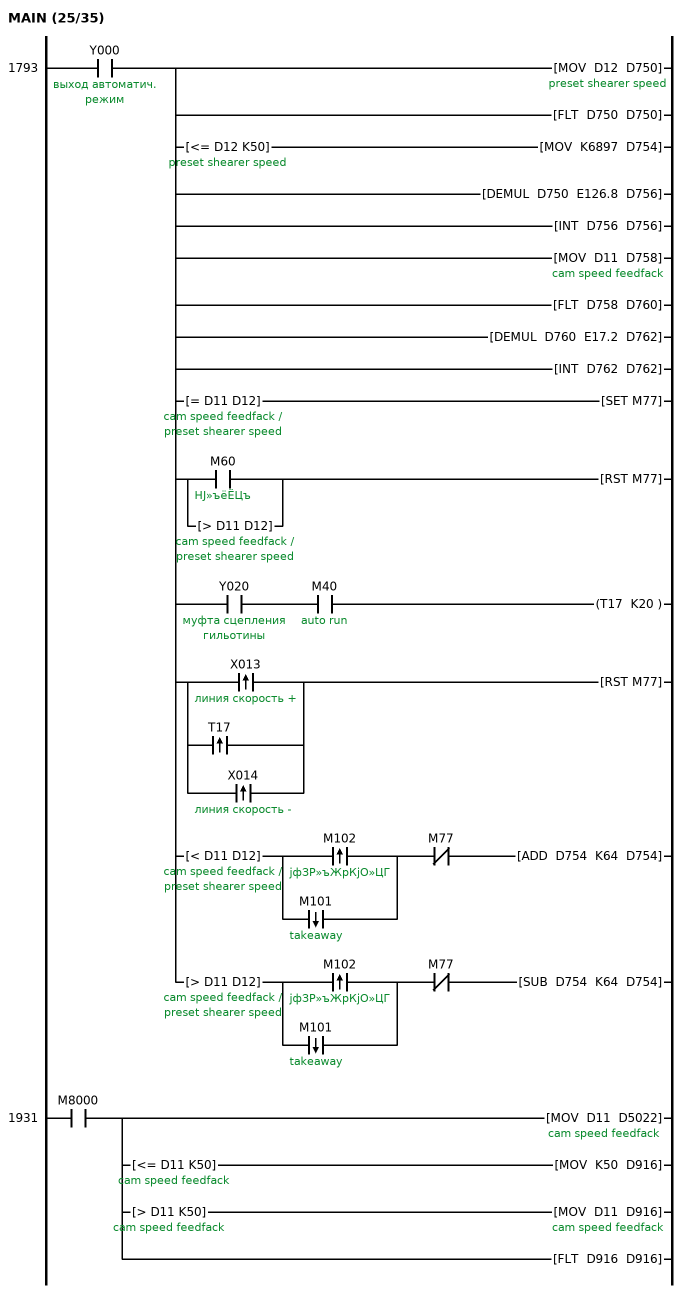
[picture p24: ladder of MAIN, rungs at steps 1793 to 1931]
1793  LD      Y000  ; выход автоматич. режим
      MOV     D12 D750
      FLT     D750 D750
      MPS
      AND<=   D12 K50  ; preset shearer speed
      MOV     K6897 D754
      MPP
      DEMUL   D750 E126.8 D756
      INT     D756 D756
      MOV     D11 D758
      FLT     D758 D760
      DEMUL   D760 E17.2 D762
      INT     D762 D762
      MPS
      AND=    D11 D12  ; cam speed feedfack / preset shearer speed
      SET     M77
      MRD
      LD      M60  ; НЈ»ъёЁЦъ
      OR>     D11 D12  ; cam speed feedfack / preset shearer speed
      ANB
      RST     M77
      MRD
      AND     Y020  ; муфта сцепления гильотины
      AND     M40  ; auto run
      OUT     T17 K20
      MRD
      LDP     X013  ; линия скорость +
      ORP     T17
      ORP     X014  ; линия скорость -
      ANB
      RST     M77
      MRD
      AND<    D11 D12  ; cam speed feedfack / preset shearer speed
      LDP     M102  ; јфЗР»ъЖрКјО»ЦГ
      ORF     M101  ; takeaway
      ANB
      ANI     M77
      ADD     D754 K64 D754
      MPP
      AND>    D11 D12  ; cam speed feedfack / preset shearer speed
      LDP     M102  ; јфЗР»ъЖрКјО»ЦГ
      ORF     M101  ; takeaway
      ANB
      ANI     M77
      SUB     D754 K64 D754
1931  LD      M8000
      MOV     D11 D5022
      MPS
      AND<=   D11 K50  ; cam speed feedfack
      MOV     K50 D916
      MRD
      AND>    D11 K50  ; cam speed feedfack
      MOV     D11 D916
      MPP
      FLT     D916 D916
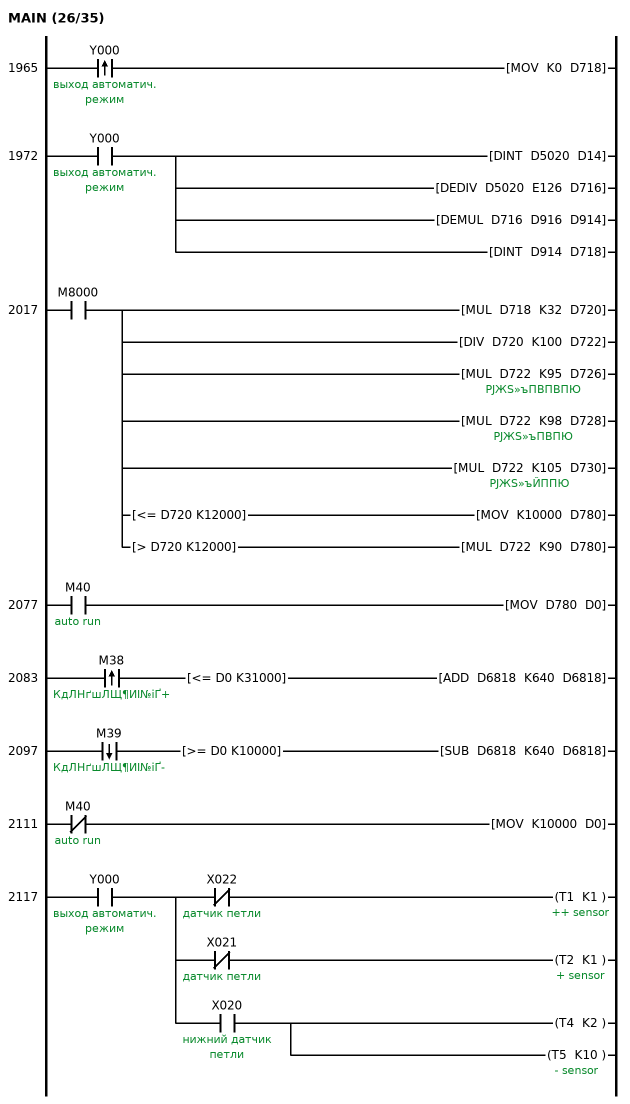
1965  LDP     Y000  ; выход автоматич. режим
      MOV     K0 D718
1972  LD      Y000  ; выход автоматич. режим
      DINT    D5020 D14
      DEDIV   D5020 E126 D716
      DEMUL   D716 D916 D914
      DINT    D914 D718
2017  LD      M8000
      MUL     D718 K32 D720
      DIV     D720 K100 D722
      MUL     D722 K95 D726  ; РЈЖЅ»ъПВПВПЮ
      MUL     D722 K98 D728  ; РЈЖЅ»ъПВПЮ
      MUL     D722 K105 D730  ; РЈЖЅ»ъЙППЮ
      MPS
      AND<=   D720 K12000
      MOV     K10000 D780
      MPP
      AND>    D720 K12000
      MUL     D722 K90 D780
2077  LD      M40  ; auto run
      MOV     D780 D0
2083  LDP     M38  ; КдЛНґшЛЩ¶ИІ№іҐ+
      AND<=   D0 K31000
      ADD     D6818 K640 D6818
2097  LDF     M39  ; КдЛНґшЛЩ¶ИІ№іҐ-
      AND>=   D0 K10000
      SUB     D6818 K640 D6818
2111  LDI     M40  ; auto run
      MOV     K10000 D0
2117  LD      Y000  ; выход автоматич. режим
      MPS
      ANI     X022  ; датчик петли
      OUT     T1 K1  ; ++ sensor
      MRD
      ANI     X021  ; датчик петли
      OUT     T2 K1  ; + sensor
      MPP
      AND     X020  ; нижний датчик петли
      OUT     T4 K2
      OUT     T5 K10  ; - sensor
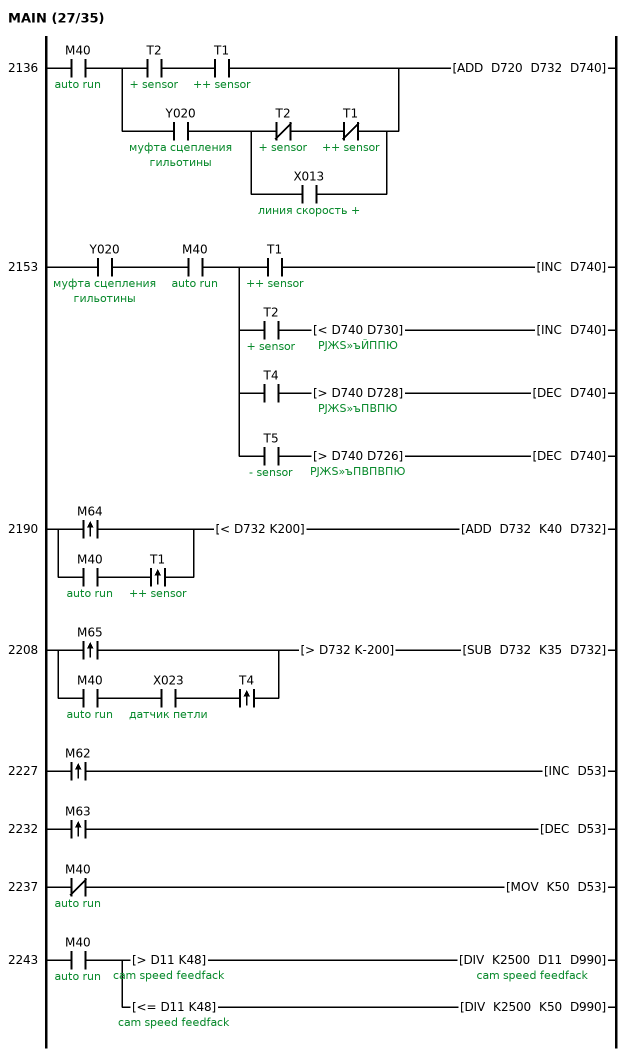
2136  LD      M40  ; auto run
      LD      T2  ; + sensor
      AND     T1  ; ++ sensor
      LD      Y020  ; муфта сцепления гильотины
      LDI     T2  ; + sensor
      ANI     T1  ; ++ sensor
      OR      X013  ; линия скорость +
      ANB
      ORB
      ANB
      ADD     D720 D732 D740
2153  LD      Y020  ; муфта сцепления гильотины
      AND     M40  ; auto run
      MPS
      AND     T1  ; ++ sensor
      INC     D740
      MRD
      AND     T2  ; + sensor
      AND<    D740 D730  ; РЈЖЅ»ъЙППЮ
      INC     D740
      MRD
      AND     T4
      AND>    D740 D728  ; РЈЖЅ»ъПВПЮ
      DEC     D740
      MPP
      AND     T5  ; - sensor
      AND>    D740 D726  ; РЈЖЅ»ъПВПВПЮ
      DEC     D740
2190  LDP     M64
      LD      M40  ; auto run
      ANDP    T1  ; ++ sensor
      ORB
      AND<    D732 K200
      ADD     D732 K40 D732
2208  LDP     M65
      LD      M40  ; auto run
      AND     X023  ; датчик петли
      ANDP    T4
      ORB
      AND>    D732 K-200
      SUB     D732 K35 D732
2227  LDP     M62
      INC     D53
2232  LDP     M63
      DEC     D53
2237  LDI     M40  ; auto run
      MOV     K50 D53
2243  LD      M40  ; auto run
      MPS
      AND>    D11 K48  ; cam speed feedfack
      DIV     K2500 D11 D990
      MPP
      AND<=   D11 K48  ; cam speed feedfack
      DIV     K2500 K50 D990
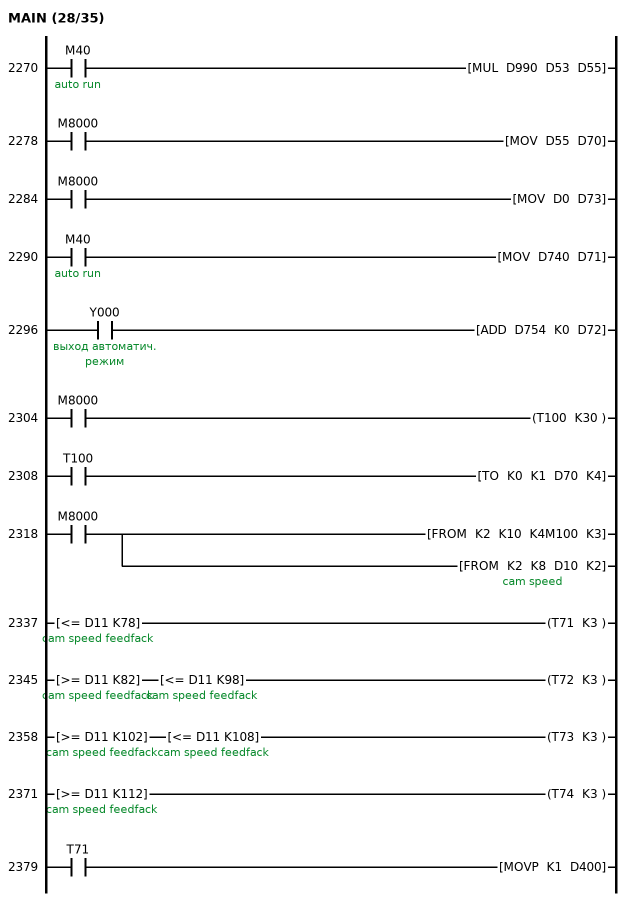
2270  LD      M40  ; auto run
      MUL     D990 D53 D55
2278  LD      M8000
      MOV     D55 D70
2284  LD      M8000
      MOV     D0 D73
2290  LD      M40  ; auto run
      MOV     D740 D71
2296  LD      Y000  ; выход автоматич. режим
      ADD     D754 K0 D72
2304  LD      M8000
      OUT     T100 K30
2308  LD      T100
      TO      K0 K1 D70 K4
2318  LD      M8000
      FROM    K2 K10 K4M100 K3
      FROM    K2 K8 D10 K2  ; cam speed
2337  LD<=    D11 K78  ; cam speed feedfack
      OUT     T71 K3
2345  LD>=    D11 K82  ; cam speed feedfack
      AND<=   D11 K98  ; cam speed feedfack
      OUT     T72 K3
2358  LD>=    D11 K102  ; cam speed feedfack
      AND<=   D11 K108  ; cam speed feedfack
      OUT     T73 K3
2371  LD>=    D11 K112  ; cam speed feedfack
      OUT     T74 K3
2379  LD      T71
      MOVP    K1 D400
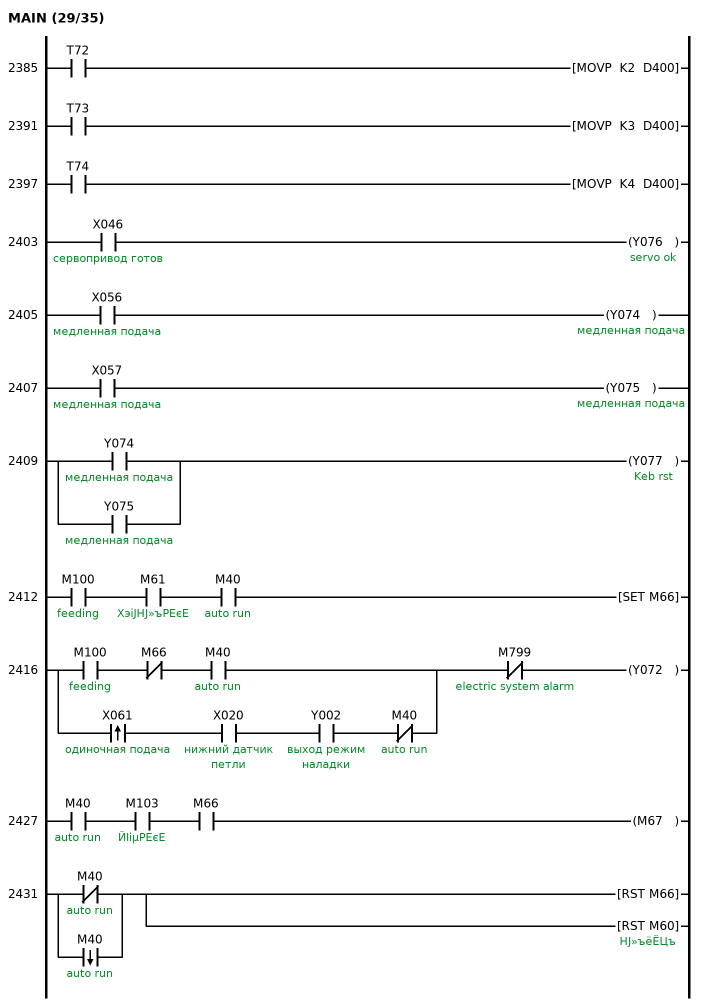
2385  LD      T72
      MOVP    K2 D400
2391  LD      T73
      MOVP    K3 D400
2397  LD      T74
      MOVP    K4 D400
2403  LD      X046  ; сервопривод готов
      OUT     Y076  ; servo ok
2405  LD      X056  ; медленная подача
      OUT     Y074  ; медленная подача
2407  LD      X057  ; медленная подача
      OUT     Y075  ; медленная подача
2409  LD      Y074  ; медленная подача
      OR      Y075  ; медленная подача
      OUT     Y077  ; Keb rst
2412  LD      M100  ; feeding
      AND     M61  ; ХэіЈНЈ»ъРЕєЕ
      AND     M40  ; auto run
      SET     M66
2416  LD      M100  ; feeding
      ANI     M66
      AND     M40  ; auto run
      LDP     X061  ; одиночная подача
      AND     X020  ; нижний датчик петли
      AND     Y002  ; выход режим наладки
      ANI     M40  ; auto run
      ORB
      ANI     M799  ; electric system alarm
      OUT     Y072
2427  LD      M40  ; auto run
      AND     M103  ; ЙІіµРЕєЕ
      AND     M66
      OUT     M67
2431  LDI     M40  ; auto run
      ORF     M40  ; auto run
      RST     M66
      RST     M60  ; НЈ»ъёЁЦъ
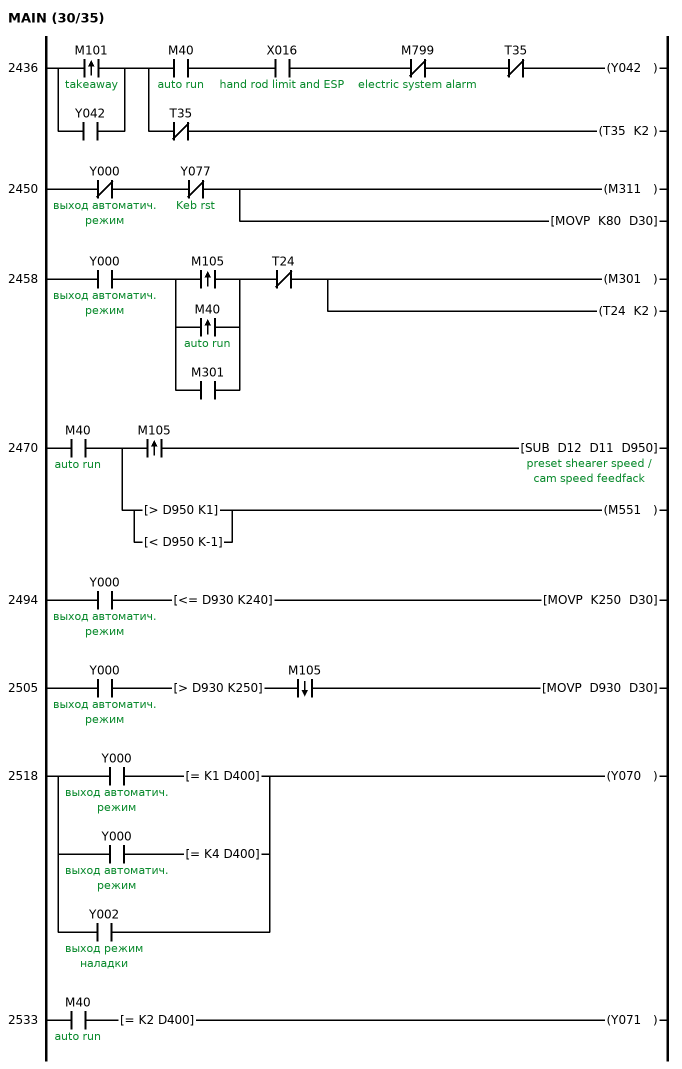
2436  LDP     M101  ; takeaway
      OR      Y042
      MPS
      AND     M40  ; auto run
      AND     X016  ; hand rod limit and ESP
      ANI     M799  ; electric system alarm
      ANI     T35
      OUT     Y042
      MPP
      ANI     T35
      OUT     T35 K2
2450  LDI     Y000  ; выход автоматич. режим
      ANI     Y077  ; Keb rst
      OUT     M311
      MOVP    K80 D30
2458  LD      Y000  ; выход автоматич. режим
      LDP     M105
      ORP     M40  ; auto run
      OR      M301
      ANB
      ANI     T24
      OUT     M301
      OUT     T24 K2
2470  LD      M40  ; auto run
      MPS
      ANDP    M105
      SUB     D12 D11 D950
      MPP
      LD>     D950 K1
      OR<     D950 K-1
      ANB
      OUT     M551
2494  LD      Y000  ; выход автоматич. режим
      AND<=   D930 K240
      MOVP    K250 D30
2505  LD      Y000  ; выход автоматич. режим
      AND>    D930 K250
      ANDF    M105
      MOVP    D930 D30
2518  LD      Y000  ; выход автоматич. режим
      AND=    K1 D400
      LD      Y000  ; выход автоматич. режим
      AND=    K4 D400
      ORB
      OR      Y002  ; выход режим наладки
      OUT     Y070
2533  LD      M40  ; auto run
      AND=    K2 D400
      OUT     Y071
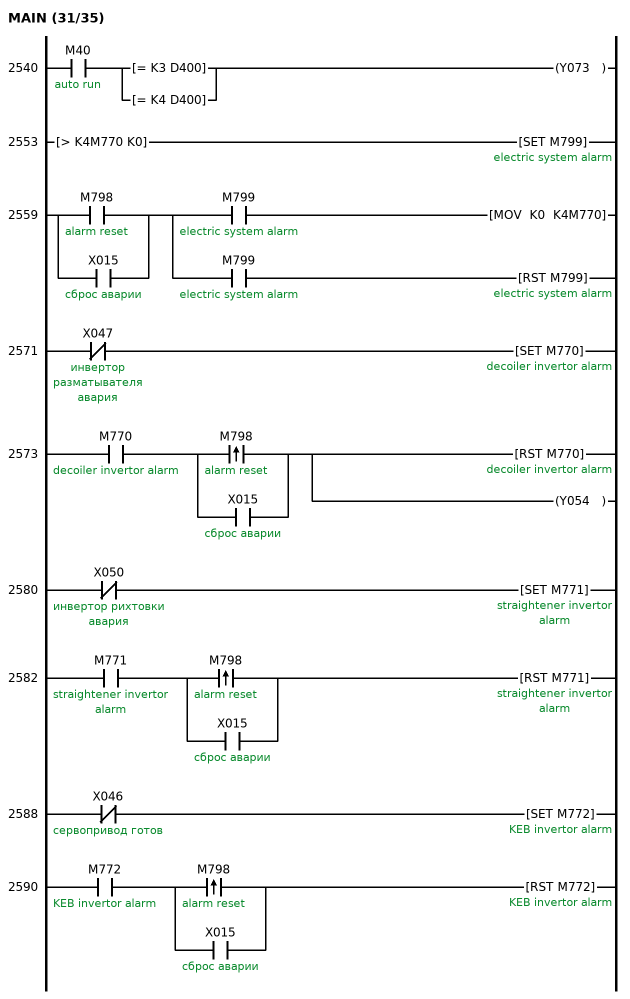
2540  LD      M40  ; auto run
      LD=     K3 D400
      OR=     K4 D400
      ANB
      OUT     Y073
2553  LD>     K4M770 K0  ; decoiler invertor alarm
      SET     M799  ; electric system alarm
2559  LD      M798  ; alarm reset
      OR      X015  ; сброс аварии
      MPS
      AND     M799  ; electric system alarm
      MOV     K0 K4M770
      MPP
      AND     M799  ; electric system alarm
      RST     M799  ; electric system alarm
2571  LDI     X047  ; инвертор разматывателя авария
      SET     M770  ; decoiler invertor alarm
2573  LD      M770  ; decoiler invertor alarm
      LDP     M798  ; alarm reset
      OR      X015  ; сброс аварии
      ANB
      RST     M770  ; decoiler invertor alarm
      OUT     Y054
2580  LDI     X050  ; инвертор рихтовки авария
      SET     M771  ; straightener invertor alarm
2582  LD      M771  ; straightener invertor alarm
      LDP     M798  ; alarm reset
      OR      X015  ; сброс аварии
      ANB
      RST     M771  ; straightener invertor alarm
2588  LDI     X046  ; сервопривод готов
      SET     M772  ; KEB invertor alarm
2590  LD      M772  ; KEB invertor alarm
      LDP     M798  ; alarm reset
      OR      X015  ; сброс аварии
      ANB
      RST     M772  ; KEB invertor alarm
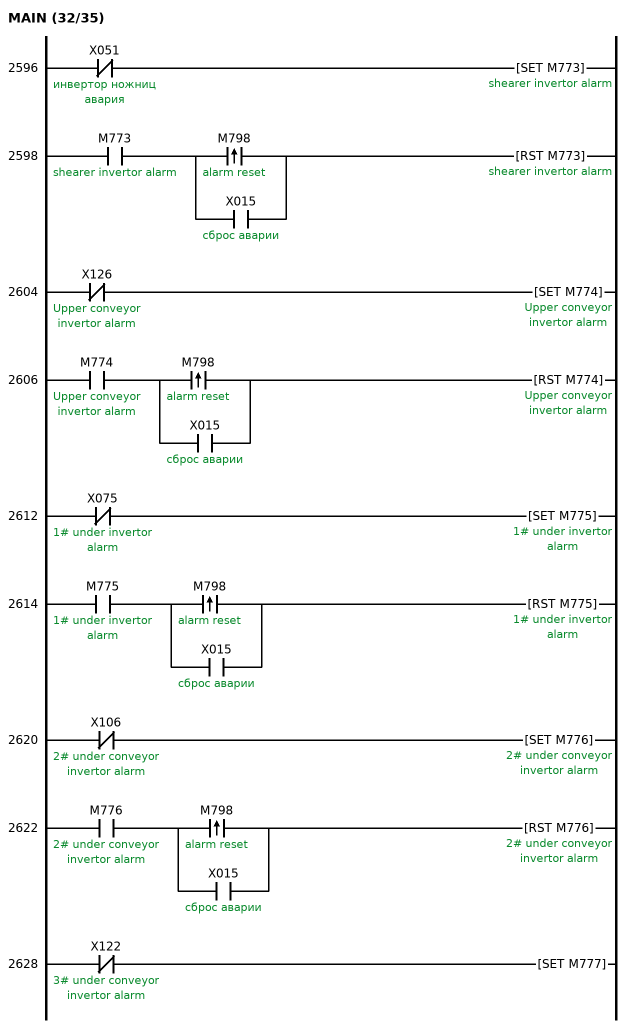
2596  LDI     X051  ; инвертор ножниц авария
      SET     M773  ; shearer invertor alarm
2598  LD      M773  ; shearer invertor alarm
      LDP     M798  ; alarm reset
      OR      X015  ; сброс аварии
      ANB
      RST     M773  ; shearer invertor alarm
2604  LDI     X126  ; Upper conveyor invertor alarm
      SET     M774  ; Upper conveyor invertor alarm
2606  LD      M774  ; Upper conveyor invertor alarm
      LDP     M798  ; alarm reset
      OR      X015  ; сброс аварии
      ANB
      RST     M774  ; Upper conveyor invertor alarm
2612  LDI     X075  ; 1# under invertor alarm
      SET     M775  ; 1# under invertor alarm
2614  LD      M775  ; 1# under invertor alarm
      LDP     M798  ; alarm reset
      OR      X015  ; сброс аварии
      ANB
      RST     M775  ; 1# under invertor alarm
2620  LDI     X106  ; 2# under conveyor invertor alarm
      SET     M776  ; 2# under conveyor invertor alarm
2622  LD      M776  ; 2# under conveyor invertor alarm
      LDP     M798  ; alarm reset
      OR      X015  ; сброс аварии
      ANB
      RST     M776  ; 2# under conveyor invertor alarm
2628  LDI     X122  ; 3# under conveyor invertor alarm
      SET     M777
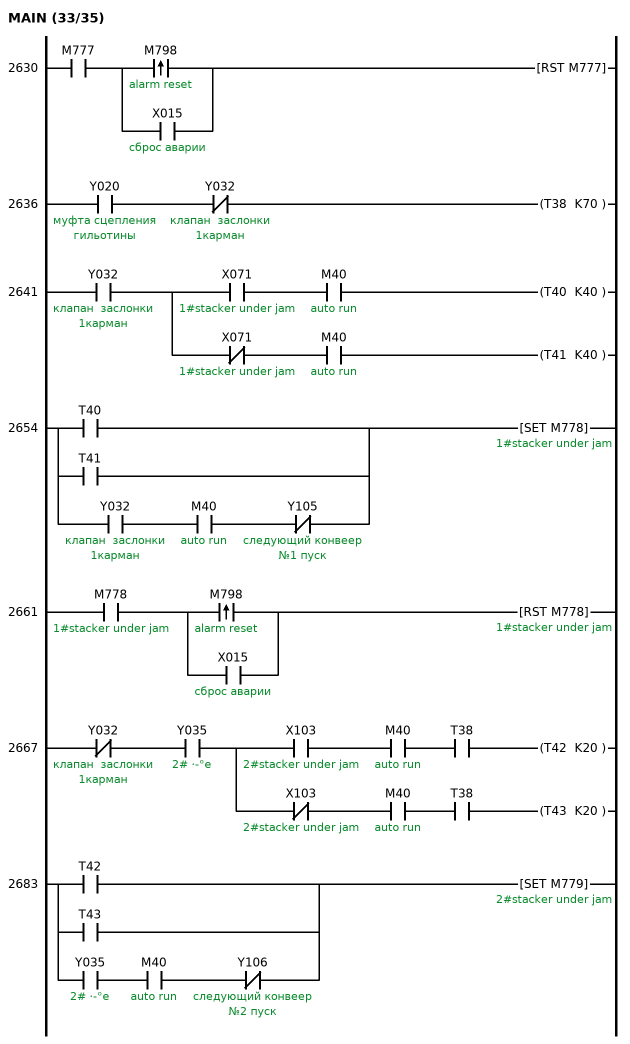
2630  LD      M777
      LDP     M798  ; alarm reset
      OR      X015  ; сброс аварии
      ANB
      RST     M777
2636  LD      Y020  ; муфта сцепления гильотины
      ANI     Y032  ; клапан  заслонки 1карман
      OUT     T38 K70
2641  LD      Y032  ; клапан  заслонки 1карман
      MPS
      AND     X071  ; 1#stacker under jam
      AND     M40  ; auto run
      OUT     T40 K40
      MPP
      ANI     X071  ; 1#stacker under jam
      AND     M40  ; auto run
      OUT     T41 K40
2654  LD      T40
      OR      T41
      LD      Y032  ; клапан  заслонки 1карман
      AND     M40  ; auto run
      ANI     Y105  ; следующий конвеер №1 пуск
      ORB
      SET     M778  ; 1#stacker under jam
2661  LD      M778  ; 1#stacker under jam
      LDP     M798  ; alarm reset
      OR      X015  ; сброс аварии
      ANB
      RST     M778  ; 1#stacker under jam
2667  LDI     Y032  ; клапан  заслонки 1карман
      AND     Y035  ; 2# ·­°е
      MPS
      AND     X103  ; 2#stacker under jam
      AND     M40  ; auto run
      AND     T38
      OUT     T42 K20
      MPP
      ANI     X103  ; 2#stacker under jam
      AND     M40  ; auto run
      AND     T38
      OUT     T43 K20
2683  LD      T42
      OR      T43
      LD      Y035  ; 2# ·­°е
      AND     M40  ; auto run
      ANI     Y106  ; следующий конвеер №2 пуск
      ORB
      SET     M779  ; 2#stacker under jam
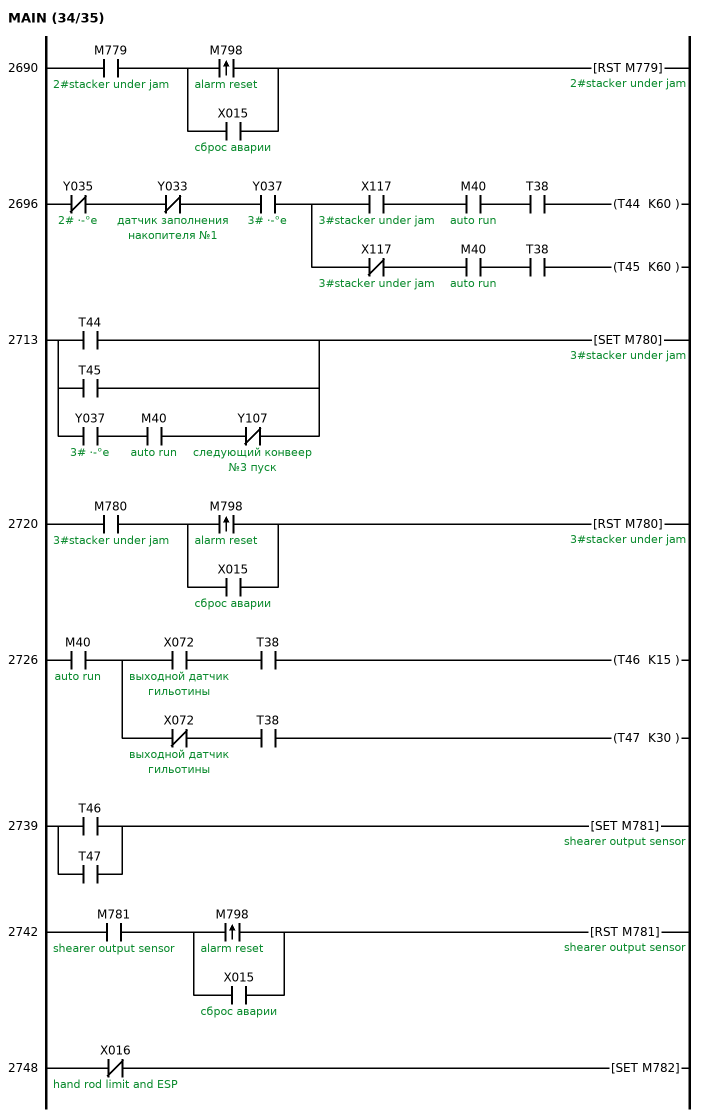
2690  LD      M779  ; 2#stacker under jam
      LDP     M798  ; alarm reset
      OR      X015  ; сброс аварии
      ANB
      RST     M779  ; 2#stacker under jam
2696  LDI     Y035  ; 2# ·­°е
      ANI     Y033  ; датчик заполнения накопителя №1
      AND     Y037  ; 3# ·­°е
      MPS
      AND     X117  ; 3#stacker under jam
      AND     M40  ; auto run
      AND     T38
      OUT     T44 K60
      MPP
      ANI     X117  ; 3#stacker under jam
      AND     M40  ; auto run
      AND     T38
      OUT     T45 K60
2713  LD      T44
      OR      T45
      LD      Y037  ; 3# ·­°е
      AND     M40  ; auto run
      ANI     Y107  ; следующий конвеер №3 пуск
      ORB
      SET     M780  ; 3#stacker under jam
2720  LD      M780  ; 3#stacker under jam
      LDP     M798  ; alarm reset
      OR      X015  ; сброс аварии
      ANB
      RST     M780  ; 3#stacker under jam
2726  LD      M40  ; auto run
      MPS
      AND     X072  ; выходной датчик гильотины
      AND     T38
      OUT     T46 K15
      MPP
      ANI     X072  ; выходной датчик гильотины
      AND     T38
      OUT     T47 K30
2739  LD      T46
      OR      T47
      SET     M781  ; shearer output sensor
2742  LD      M781  ; shearer output sensor
      LDP     M798  ; alarm reset
      OR      X015  ; сброс аварии
      ANB
      RST     M781  ; shearer output sensor
2748  LDI     X016  ; hand rod limit and ESP
      SET     M782
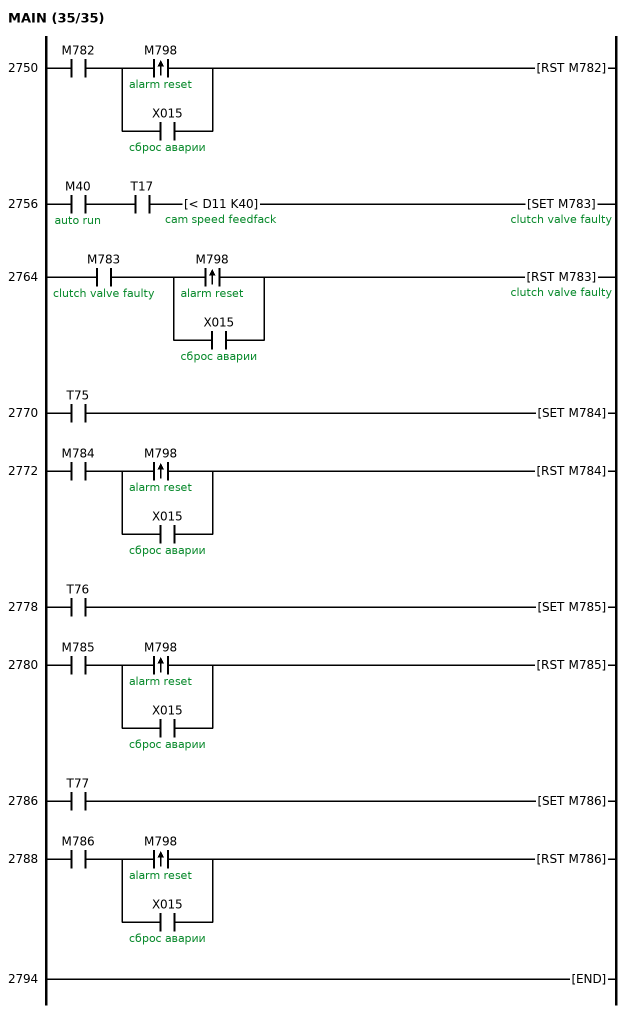
2750  LD      M782
      LDP     M798  ; alarm reset
      OR      X015  ; сброс аварии
      ANB
      RST     M782
2756  LD      M40  ; auto run
      AND     T17
      AND<    D11 K40  ; cam speed feedfack
      SET     M783  ; clutch valve faulty
2764  LD      M783  ; clutch valve faulty
      LDP     M798  ; alarm reset
      OR      X015  ; сброс аварии
      ANB
      RST     M783  ; clutch valve faulty
2770  LD      T75
      SET     M784
2772  LD      M784
      LDP     M798  ; alarm reset
      OR      X015  ; сброс аварии
      ANB
      RST     M784
2778  LD      T76
      SET     M785
2780  LD      M785
      LDP     M798  ; alarm reset
      OR      X015  ; сброс аварии
      ANB
      RST     M785
2786  LD      T77
      SET     M786
2788  LD      M786
      LDP     M798  ; alarm reset
      OR      X015  ; сброс аварии
      ANB
      RST     M786
2794  END
END_PROGRAM

// device comments not shown above
X026  ; aid support limit
X127  ; none
Y021  ; сигнал заполнения накопителя №1
D1  ; РЈЖЅ»ъЛЩ¶ИКдіц
D2  ; јфЗР»ъЛЩ¶ИКдіц
D3  ; ЙПєу¶ОКдЛНґшЛЩ¶И
